{attribute addProperty BoxType "EJ5002-0000-0017"}
{attribute addProperty Id "StatusAT %I*Status_F6CF9E121621Counter_valueAT %I*UDINT32417"}
{attribute addProperty CRC "851906893"}
{attribute addProperty SizeInBites "48"}
{attribute addProperty SizeInBytes "6"}
TYPE SSI_Inputs_Channel_32C7114D :
STRUCT
	{attribute addProperty Name "Status"}
	Status AT %I* : Status_F6CF9E12;
	{attribute addProperty Name "Counter_value"}
	Counter_value AT %I* : UDINT;
END_STRUCT
END_TYPE

(* stored: Version 1.2.0.0, ProductVersion 3.1.4024.9
   DUT SSI_Inputs_Channel_32C7114D: Id {9f8c3ef9-3d14-4975-9ca3-7086ff8b88fd} *)
